// TIA Portal V17 export
// export: Created 2023-05-07T12:12:21.6102017Z, ExportSetting WithDefaults, DisplayName Totally Integrated Automation Portal, DisplayVersion V17, DisplayName TIA Portal Openness, DisplayVersion V17, DisplayName TIA Portal Version Control Interface, DisplayVersion V17, DisplayName TIA Portal Test Suite Advanced, DisplayVersion V17, DisplayName STEP 7 Professional, DisplayVersion V17, DisplayName SIMATIC Energy Suite, DisplayVersion V17, DisplayName STEP 7 Safety, DisplayVersion V17, DisplayName WinCC Professional, DisplayVersion V17
FUNCTION "DisturbanceClass" : Void   // FC5, LAD
TITLE = DisturbanceClass
{ S7_Optimized_Access := 'TRUE' }
VERSION : 0.1
// stored: AutoNumber true, IsIECCheckEnabled false, SetENOAutomatically false, UDAEnableTagReadback false
   VAR_TEMP
      MV : Real;
   END_VAR
BEGIN

REGION Network 1: Call: RandomDisturbance
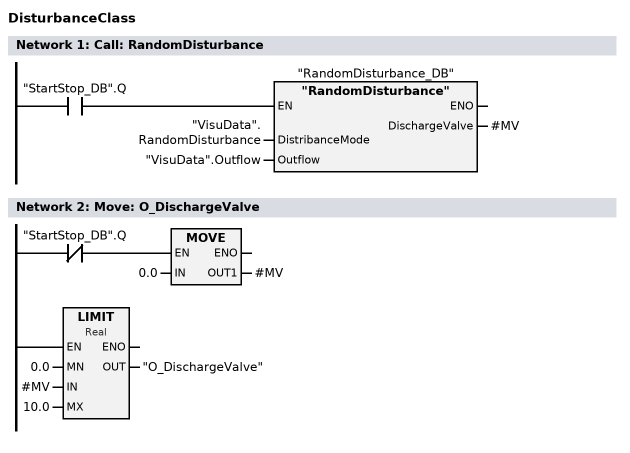
   RUNG wire#powerrail
      Contact( "StartStop_DB".Q )
      "RandomDisturbance_DB"(DistribanceMode := "VisuData".RandomDisturbance, Outflow := "VisuData".Outflow, DischargeValve => #MV)
   END_RUNG
   // the same network as SCL:
   IF "StartStop_DB".Q THEN
       "RandomDisturbance_DB"(DistribanceMode := "VisuData".RandomDisturbance,   // "RandomDisturbance"
                              Outflow := "VisuData".Outflow,
                              DischargeValve => #MV);
   END_IF;
END_REGION

REGION Network 2: Move: O_DischargeValve
   RUNG wire#powerrail
      I_Contact( "StartStop_DB".Q )
      Move(in := 0.0, out1 => #MV)
   END_RUNG
   RUNG wire#powerrail
      { S7_Templates := "value_type := Real" } Limit(mn := 0.0, in := #MV, mx := 10.0, out => "O_DischargeValve")
   END_RUNG
   // the same network as SCL:
   IF NOT "StartStop_DB".Q THEN #MV := 0.0; END_IF;
   "O_DischargeValve" := LIMIT(MN := 0.0, IN := #MV, MX := 10.0);
END_REGION
END_FUNCTION
